{attribute 'GeneratedUsingTerminal: EK1100-0000-0018'}
{attribute addProperty BoxType "EK1100-0000-0018"}
{attribute addProperty Id "Beckhoff_EPP4xxxEK1122Beckhoff_EPP4xxxEK1122_C4216F90222"}
{attribute addProperty CRC "2842134423"}
{attribute addProperty Size "222"}
TYPE Beckhoff_EPP4xxx_A9678797 EXTENDS EK1100_1FC0878B :
STRUCT
	{attribute addProperty Name "Beckhoff_EPP4xxxEK1122"}
	{attribute addProperty PreviousPort "Beckhoff EPP4xxx : B"}
	Beckhoff_EPP4xxxEK1122 : Beckhoff_EPP4xxxEK1122_C4216F90;
END_STRUCT
END_TYPE

(* stored: Version 1.2.0.0, ProductVersion 3.1.4024.9
   DUT Beckhoff_EPP4xxx_A9678797: Id {afa54044-a744-457f-a66c-f84de0abf22f} *)
